FUNCTION_BLOCK RunningUnifiedProgramState EXTENDS RunningProgramState
VAR_STAT
	//! <summary>Class name shared by all instances of this function block.</summary>
	{attribute 'OPC.UA.DA' := '0'}
	_ClassName : STRING := __POUNAME();
END_VAR

{attribute 'monitoring' := 'call'}
PROPERTY ClassName : REFERENCE TO STRING
GET
ClassName REF= _ClassName;
END_GET
END_PROPERTY

END_FUNCTION_BLOCK

(* stored: Version 1.1.0.1
   POU RunningUnifiedProgramState: Id {4b251c1d-0adf-42da-bd3c-c3415ff180f8}, SpecialFunc None
   Property ClassName: Id {29bf2687-06c2-46dd-b807-62acad5530e1}
   Get Get: Id {0877b4ac-7155-4bf2-8f14-afc82558813f} *)
